// TIA Portal V17 export
// export: Created 2024-09-02T12:50:18.2024097Z, ExportSetting WithDefaults, DisplayName Totally Integrated Automation Portal, DisplayVersion V17, DisplayName TIA Portal Openness, DisplayVersion V17, DisplayName TIA Portal Version Control Interface, DisplayVersion V17, DisplayName STEP 7 Professional, DisplayVersion V17, DisplayName STEP 7 Safety, DisplayVersion V17, DisplayName WinCC Professional, DisplayVersion V17
DATA_BLOCK "LTLL_ManualGraphControl_OP70"   // DB464
TITLE = LTLL_ManualGraphControl
{ S7_Optimized_Access := 'TRUE'; DB_Accessible_From_OPC_UA := 'FALSE' }
AUTHOR : Siemens
FAMILY : HMI_Lite
NAME : LTLL_ManualGraphControl
VERSION : 8.10
// stored: AutoNumber true, DBAccessibleFromOPCUA false, InstanceOfName LTLL_typeManualGraphControl, InstanceOfType UDT, IsOnlyStoredInLoadMemory false, IsWriteProtectedInAS false
"LTLL_typeManualGraphControl"
   // VAR
   //    screen { S7_SetPoint := 'True'} : Array[0..6] of "LTLL_typeGraphControl";
   // END_VAR
BEGIN
END_DATA_BLOCK
